TYPE ST_MaterialDataX :
STRUCT
	{attribute 'OPC.UA.DA.Description' := 'Job data type'}

END_STRUCT
END_TYPE

(* stored: Version 1.1.0.1, ProductVersion 3.1.4024.5
   DUT ST_MaterialDataX: Id {477320ea-9047-4d38-8c8a-15348eee0cf3} *)
